TYPE Room_Settings_PassiveTempTime :
STRUCT
	timee			: Room_Settings_TimeSettings;
	temp			: Room_Settings_TemperatureSettings;
	bEnablePassive	: BOOL;
END_STRUCT
END_TYPE

(* stored: Version 1.1.0.1
   DUT Room_Settings_PassiveTempTime: Id {fa04fa4b-335f-4506-b254-d545b968b9df} *)
